TYPE AxisFn :
STRUCT
	MC_Power		: MC_Power;
	MC_Reset		: MC_Reset;
	MC_SetPosition	: MC_SetPosition;
END_STRUCT
END_TYPE

(* stored: Version 1.1.0.1, ProductVersion 3.1.4022.17
   DUT AxisFn: Id {2daf280a-653d-4079-8b06-cc9aee314ec8} *)
